TYPE ST_EC_SIM_Device_Inputs :
STRUCT
	Status							:UDINT;
	Telegram_Counter				:UDINT;
	Dc_Time							:ULINT;
	Dc_Time_to_System_Time_Offset	:ULINT;
	{attribute 'displaymode':='hex'} 
	DevState						:UINT;
	AmsNetId						:AMSNETID;
END_STRUCT
END_TYPE

(* stored: Version 1.1.0.1, ProductVersion 3.1.4024.11
   DUT ST_EC_SIM_Device_Inputs: Id {abd9f4f1-66f4-4905-b091-ede4231214f8} *)
